// TIA Portal V20 export
TYPE "typeInterfaceSignalsHmi"
TITLE = Schnittstellen Signale HMI / Interface signals HMI
// Struktur Schnittstelle Signale fuer HMI / Structure interface signals Bool HMI
// stored: Access Published
   STRUCT
      valueSymbolLeft : "LAF_typeInterfaceSignalsBool";   // Werte Symbol links / Value symbol lleft
      valueSymbolRight : "LAF_typeInterfaceSignalsBool";   // Werte Symbol rechts / Value symbol rght
   END_STRUCT;
END_TYPE
